Staubli VAL3: init_prgm.pgx

public program init_prgm()
begin

  // mise en rotation pompe vitesse nulle
    aioSet(Tpompe,0)
    put("Pompe en rotation")
    // arrêt pompe
    dioSet(doPompe,0)
    put("Pompe arret")
    // fermeture obturateur
    dioSet(doValve2,0)
    dioSet(doValve1,1)
    put("Obturateur fermé")

end
